(* CODESYS project Accumulator_Rev1.0.0.260412.project

Project tree, tasks and I/O mapping:
  PLCWinNT : CODESYS Control Win V3, CODESYS, version 3.5.22.0
    application Application
      libraries: Standard, * (System)
      task MainTask (cyclic, interval t#50ms, priority 1) calls PLC_PRG
      program PLC_PRG [ST]
      global variables GVL_Accumulator
*)

// PLCWinNT/Application/GVL_Accumulator
VAR_GLOBAL
    g_nAccumulator : INT := 0;
    g_nCycleCount : DINT := 0;
    g_bEnable : BOOL := TRUE;
    g_nStep : INT := 1;
    g_nMaxValue : INT := 1000;
END_VAR

// PLCWinNT/Application/PLC_PRG
PROGRAM PLC_PRG
VAR
    nAccumulator : INT := 0;
    nStep : INT := 1;
    nMaxValue : INT := 1000;
    nCycleCount : DINT := 0;
    bEnable : BOOL := TRUE;
    bReset : BOOL := FALSE;
END_VAR

IF bEnable THEN
    IF bReset THEN
        nAccumulator := 0;
        nCycleCount := 0;
        bReset := FALSE;
    END_IF;

    nAccumulator := nAccumulator + nStep;

    IF nAccumulator >= nMaxValue THEN
        nAccumulator := 0;
        nCycleCount := nCycleCount + 1;
    END_IF;
END_IF

END_PROGRAM
